FUNCTION_BLOCK startSorting
VAR_INPUT
    grab: grab; 
	timer : TP;	
	ccw: moveCCW;
	cw:moveCW;
	down:moveDown;
	iztegni:moveOUT;
	skrci:moveIN;
	up: moveUp;
	relise: relise; 
END_VAR
VAR_OUTPUT
	 done: BOOL := FALSE; // Indikator, da je sekvenca zaključena
END_VAR
VAR
	currentState: INT := 0; // Trenutno stanje sekvence
	
	obDol: INT;
	objekt: INT;
	itemID: INT := 1; //item number
	TimerWait: TOF;
	I: INT;
END_VAR

CASE currentState OF
    // Stanje 0: Priprava
    0:
        done := FALSE;         // Ponastavi indikator zaključka
        GVL.downDone := FALSE;     // Ponastavi zastavico za premik dol
        GVL.grabDone := FALSE;     // Ponastavi zastavico za prijem
        currentState := 1;     // Premik na naslednje stanje

    1://PREMIK DOL PO OBJEKTIH
		 //grab(seconds := T#1.5S);     // Aktiviraj prijem
		grab(seconds := T#2.2S);
        IF GVL.grabDone THEN           // Počakaj, da je prijem zaključen
            //grabDone := TRUE;       // Nastavi zastavico
            currentState := 2;      // Premik na naslednje stanje
			GVL.grabDone := FALSE;
        END_IF
		
	2:	
		ccw(seconds := T#2.5S);
			IF GVL.CCWDone THEN           // Počakaj, da je prijem zaključen
				currentState := 3;      // Premik na naslednje stanje
				GVL.CCWDone := FALSE;
			END_IF
			
	3:
		cw(seconds := T#2.5S);
        IF GVL.CWDone THEN           // Počakaj, da je prijem zaključen
            currentState := 4;      // Premik na naslednje stanje
			GVL.CWDone := FALSE;
        END_IF
	4:
		down(seconds := T#1S);  // Aktiviraj premik dol
		IF GVL.downDone THEN          // Počakaj, da je premik zaključen
			//downDone := TRUE;      // Nastavi zastavico
			currentState := 5;     // Premik na naslednje stanje
			GVL.downDone := FALSE;
		END_IF
		
	5:
		iztegni(seconds := T#1S);
        IF GVL.skrciDone THEN           // Počakaj, da je prijem zaključen
            currentState := 6;      // Premik na naslednje stanje
			GVL.skrciDone := FALSE;
        END_IF
		
	6:
		skrci(seconds := T#1S);
        IF GVL.skrciDone THEN           // Počakaj, da je prijem zaključen
            currentState := 7;      // Premik na naslednje stanje
			GVL.skrciDone := FALSE;
        END_IF
	7:
		up(seconds := T#2S);
        IF GVL.upDone THEN           // Počakaj, da je prijem zaključen
            currentState := 8;      // Premik na naslednje stanje
			GVL.upDone := FALSE;
        END_IF
	8:
		relise(seconds := T#2S);
        IF GVL.reliseDone THEN           // Počakaj, da je prijem zaključen
            currentState := 8;      // Premik na naslednje stanje
			GVL.reliseDone := FALSE;
        END_IF
	
END_CASE

END_FUNCTION_BLOCK

(* stored: Version 1.1.0.1, ProductVersion 3.1.4024.15
   POU startSorting: Id {9c246b88-e24f-4b9e-9a0d-43507cde2e96}, SpecialFunc None *)
